Yaskawa INFORM job: MCRPATH.JBI

/JOB
//NAME MCRPATH
//POS
///NPOS 0,0,0,0,0,0
//INST
///DATE 2010/10/22 10:58
///ATTR SC,RW,MC
///GROUP1 RB1
NOP
SKILLSND "corrpath"
END
